ABB RobotStudio station: Alushi_Yumi_EGM_2024.rsstnx

Station Alushi_Yumi_EGM_2024 (saved by RobotStudio 23.2.10395.0)
Controller YuMi_EGM_Alushi_2024, task T_ROB_L: task frame (RAPID world) sits at (-150, 0, 308) mm in the station
Controller YuMi_EGM_Alushi_2024, task T_ROB_R: task frame (RAPID world) sits at (-150, 0, 308) mm in the station
Controller YuMi_EGM_Alushi_2024
  mechanical unit ROB_R: IRB14000_0.5_0.5_R, 6 joints, base frame (0, 0, 0) mm
  mechanical unit ROB_R_7: IRB14000_0.5_0.5_R, 1 joints, base frame (0, 0, 0) mm
  mechanical unit ROB_L: IRB14000_0.5_0.5_L, 6 joints, base frame (0, 0, 0) mm
  mechanical unit ROB_L_7: IRB14000_0.5_0.5_L, 1 joints, base frame (0, 0, 0) mm
Layout (positions relative to the parent item):
  - table [part] at (175, -225, 0) mm, rotated rx 0 ry 0 rz 90 deg, size 450 x 350 x 308 mm
  - IRB14000_0.5_0.5 [mechanism, from %ABB.RobotStudio.Models.IRB14000%\IRB14000_0.5_0.5__02.rslib] at (-150, 0, 308) mm
  - IRB14000_0.5_0.5_R [mechanism, from %ABB.RobotStudio.Models.IRB14000%\IRB14000_0.5_0.5__02.rslib] at (-150, 0, 308) mm; joint values [0, -2.2689, -2.3562, 0.5236, 0, 0.6981, 0] (rad or m)
  - IRB14000_0.5_0.5_L [mechanism, from %ABB.RobotStudio.Models.IRB14000%\IRB14000_0.5_0.5__02.rslib] at (-150, 0, 308) mm; joint values [2.5625, 0.2936, 0.766, 0.4369, -1.9215, 0.653, 0.9137] (rad or m)
Targets, tools, work objects and paths stored in the station, written as RAPID:
! task T_ROB_R
MODULE Module_Right_Arm_IRB14000
  PROC main()
    MoveAbsJ joints,v1000,fine,tool0;
    StartEGM;
    WaitTime 1;
  ENDPROC
  PROC StartEGM()
  ENDPROC
ENDMODULE

! task T_ROB_L
MODULE Module_Left_Arm_IRB14000
  PROC main()
    MoveAbsJ joints,v1000,fine,tool0;
    StartEGM;
    WaitTime 1;
  ENDPROC
  PROC StartEGM()
  ENDPROC
ENDMODULE

